// TwinCAT 3 PLC project plc
// ProgramVersion: 3.1.4024.0
// libraries:
//   Tc2_Standard, * (Beckhoff Automation GmbH)
//   Tc2_System, * (Beckhoff Automation GmbH)
//   Tc3_Module, * (Beckhoff Automation GmbH)
// project tree:
//   DUTs/ Axis_OUTPUT.TcDUT, Axis_STATUS.TcDUT
//   / PlcTask.TcTTO (not stored)
//   POUs/ MAIN.TcPOU
// real-time tasks:
//   TASK PlcTask: cycle T#10ms, priority 20, ADS port 350
// I/O:
//   DEVICE Device 3 (EtherCAT), AmsNetId 169.254.115.184.4.1
//     Box 4 (EX1616DN) [EX1616DN]
//       modules: Module 1 (SX1616DN)
//     Drive 1 (MCDLN35BE) [MCDLN35BE]
//     Drive 2 (MCDLN35BE) [MCDLN35BE]
//     Drive 3 (MBDLN25BE) [MBDLN25BE]
// variable links:
//   plc/plc Instance <-> Device 3 (EtherCAT)/Box 4 (EX1616DN)
//     PlcTask Outputs/MAIN.BREAK0 <-> Module 1 (SX1616DN)/Outputs/Digital16 OUT
//   plc/plc Instance <-> Device 3 (EtherCAT)/Drive 1 (MCDLN35BE)
//     PlcTask Inputs/MAIN.Axis0_status/Actual_Position <-> Transmit PDO mapping 1/Position actual value
//     PlcTask Inputs/MAIN.Axis0_status/Actual_Torque <-> Transmit PDO mapping 1/Torque actual value
//     PlcTask Inputs/MAIN.Axis0_status/Actual_Velocity <-> Transmit PDO mapping 1/Velocity actual value
//     PlcTask Inputs/MAIN.Axis0_status/Following_error <-> Transmit PDO mapping 1/Following error actual value
//     PlcTask Inputs/MAIN.Axis0_status/Mode_of_Operation_disp <-> Transmit PDO mapping 1/Modes of operation display
//     PlcTask Inputs/MAIN.Axis0_status/Status <-> Transmit PDO mapping 1/Statusword
//     PlcTask Outputs/MAIN.Axis0/Control_Word <-> Receive PDO mapping 1/Controlword
//     PlcTask Outputs/MAIN.Axis0/Max_Torque <-> Receive PDO mapping 1/Max torque
//     PlcTask Outputs/MAIN.Axis0/Max_Velocity <-> Receive PDO mapping 1/Max motor speed
//     PlcTask Outputs/MAIN.Axis0/Mode_of_Operation <-> Receive PDO mapping 1/Modes of operation
//     PlcTask Outputs/MAIN.Axis0/Profile_Velocity <-> Receive PDO mapping 1/Profile velocity
//     PlcTask Outputs/MAIN.Axis0/Target_Position <-> Receive PDO mapping 1/Target position
//     PlcTask Outputs/MAIN.Axis0/Target_Torque <-> Receive PDO mapping 1/Target torque
//   plc/plc Instance <-> Device 3 (EtherCAT)/Drive 2 (MCDLN35BE)
//     PlcTask Inputs/MAIN.Axis1_status/Actual_Position <-> Transmit PDO mapping 1/Position actual value
//     PlcTask Inputs/MAIN.Axis1_status/Actual_Torque <-> Transmit PDO mapping 1/Torque actual value
//     PlcTask Inputs/MAIN.Axis1_status/Actual_Velocity <-> Transmit PDO mapping 1/Velocity actual value
//     PlcTask Inputs/MAIN.Axis1_status/Following_error <-> Transmit PDO mapping 1/Following error actual value
//     PlcTask Inputs/MAIN.Axis1_status/Mode_of_Operation_disp <-> Transmit PDO mapping 1/Modes of operation display
//     PlcTask Inputs/MAIN.Axis1_status/Status <-> Transmit PDO mapping 1/Statusword
//     PlcTask Outputs/MAIN.Axis1/Control_Word <-> Receive PDO mapping 1/Controlword
//     PlcTask Outputs/MAIN.Axis1/Max_Torque <-> Receive PDO mapping 1/Max torque
//     PlcTask Outputs/MAIN.Axis1/Max_Velocity <-> Receive PDO mapping 1/Max motor speed
//     PlcTask Outputs/MAIN.Axis1/Mode_of_Operation <-> Receive PDO mapping 1/Modes of operation
//     PlcTask Outputs/MAIN.Axis1/Profile_Velocity <-> Receive PDO mapping 1/Profile velocity
//     PlcTask Outputs/MAIN.Axis1/Target_Position <-> Receive PDO mapping 1/Target position
//     PlcTask Outputs/MAIN.Axis1/Target_Torque <-> Receive PDO mapping 1/Target torque
//   plc/plc Instance <-> Device 3 (EtherCAT)/Drive 3 (MBDLN25BE)
//     PlcTask Inputs/MAIN.Axis2_status/Actual_Position <-> Transmit PDO mapping 1/Position actual value
//     PlcTask Inputs/MAIN.Axis2_status/Actual_Torque <-> Transmit PDO mapping 1/Torque actual value
//     PlcTask Inputs/MAIN.Axis2_status/Actual_Velocity <-> Transmit PDO mapping 1/Velocity actual value
//     PlcTask Inputs/MAIN.Axis2_status/Following_error <-> Transmit PDO mapping 1/Following error actual value
//     PlcTask Inputs/MAIN.Axis2_status/Mode_of_Operation_disp <-> Transmit PDO mapping 1/Modes of operation display
//     PlcTask Inputs/MAIN.Axis2_status/Status <-> Transmit PDO mapping 1/Statusword
//     PlcTask Outputs/MAIN.Axis2/Control_Word <-> Receive PDO mapping 1/Controlword
//     PlcTask Outputs/MAIN.Axis2/Max_Torque <-> Receive PDO mapping 1/Max torque
//     PlcTask Outputs/MAIN.Axis2/Max_Velocity <-> Receive PDO mapping 1/Max motor speed
//     PlcTask Outputs/MAIN.Axis2/Mode_of_Operation <-> Receive PDO mapping 1/Modes of operation
//     PlcTask Outputs/MAIN.Axis2/Profile_Velocity <-> Receive PDO mapping 1/Profile velocity
//     PlcTask Outputs/MAIN.Axis2/Target_Position <-> Receive PDO mapping 1/Target position
//     PlcTask Outputs/MAIN.Axis2/Target_Torque <-> Receive PDO mapping 1/Target torque

// ---- DUTs/Axis_OUTPUT.TcDUT
TYPE Axis_OUTPUT :
STRUCT
	Control_Word AT%Q*:WORD;
	Target_Position AT%Q*:DINT;
	Profile_Velocity AT%Q*:UDINT;
	Max_Velocity AT%Q*:UDINT;
	Mode_of_Operation AT%Q* :BYTE:=1;
	Target_Torque AT%Q* :INT:=0;
	Max_Torque AT%Q*: UINT :=0;
END_STRUCT
END_TYPE

// ---- DUTs/Axis_STATUS.TcDUT
TYPE Axis_STATUS :
STRUCT
	Status : WORD;
	Mode_of_Operation_disp:BYTE;
	Actual_Position:DINT;
	Actual_Velocity :DINT;
	Following_error:DINT;
	Actual_Torque:INT;
END_STRUCT
END_TYPE

// ---- POUs/MAIN.TcPOU
PROGRAM MAIN
VAR
	Axis0 AT%QD0:Axis_OUTPUT;
	Axis1 AT%QD6:Axis_OUTPUT;
	Axis2 AT%QD12:Axis_OUTPUT;
	
	Axis0_status AT%ID0:Axis_STATUS;
	Axis1_status AT%ID5:Axis_STATUS;
	Axis2_status AT%ID10:Axis_STATUS;
	
	BREAK0 AT%QD100 :UINT:=0;
	
END_VAR

END_PROGRAM
